FUNCTION_BLOCK GetComponentsTaskResultVisitor IMPLEMENTS I_ComponentVisitor, I_TaskResult
VAR
	{attribute 'hide'}
	Result : I_TaskResult;
	{attribute 'hide'}
	_Busy : BOOL;
	{attribute 'hide'}
	_Error : BOOL;
	{attribute 'hide'}
	_ErrorId : UDINT;
END_VAR

{attribute 'monitoring' := 'call'}
PROPERTY Busy : BOOL
GET
Busy := _Busy;
END_GET
END_PROPERTY

{attribute 'monitoring' := 'call'}
PROPERTY Error : BOOL
GET
Error := _Error;
END_GET
END_PROPERTY

{attribute 'monitoring' := 'call'}
PROPERTY ErrorId : UDINT
GET
ErrorID := _ErrorID;
END_GET
END_PROPERTY

METHOD Update
VAR_INPUT
	Module : I_Module;
END_VAR
_Error	 := FALSE;
_ErrorId := 0;
_Busy	 := FALSE;
Module.Components.Accept(THIS^);
END_METHOD

METHOD VisitComponent
VAR_INPUT
	Component : I_Component;
END_VAR
IF __QUERYINTERFACE(Component, Result) THEN
	IF Result.Error THEN
		_Error	 := TRUE;
		_ErrorId := Result.ErrorId;
	END_IF

	IF Result.Busy THEN
		_Busy := TRUE;
	END_IF
END_IF
END_METHOD

END_FUNCTION_BLOCK

(* stored: Version 1.1.0.1, ProductVersion 3.1.4026.18
   POU GetComponentsTaskResultVisitor: Id {81e09bd7-aa71-4399-b8c1-161dd5e96b69}, SpecialFunc None
   Property Busy: Id {8a6e7cab-08ce-4238-8ab8-e67b441ca527}
   Get Get: Id {baef1af1-4e2e-4242-8562-939ef234108b}
   Property Error: Id {42d4a95e-5ded-486a-b912-b6940e69e8ea}
   Get Get: Id {fd788870-39ae-4f46-88f2-5471d086ecf5}
   Property ErrorId: Id {1822047d-b94a-4962-84ba-19bb541e9af3}
   Get Get: Id {fe90a54a-addc-47d1-b737-7a7870db260d}
   Method Update: Id {edc5af62-29cb-42a3-8bb7-217c11e1b74a}
   Method VisitComponent: Id {aef0f30d-a565-4685-be76-551948d6f8a9} *)
